// TIA Portal project "zadanie_2_Kral_dzvonar" (V15.1)

(* hardware
DEVICE "S7-1200 station_1"  S7-1200 Station
   slot 0: "Rack_0"  S7-1200 Rack  Rack  V1.0
   slot 1: "PLC_1"  CPU 1215C DC/DC/DC  6ES7 215-1AG40-0XB0  V4.3
*)

// ===== PLC "PLC_1"  CPU 1215C DC/DC/DC =====

VAR_GLOBAL   // PLC tag table "Default tag table"
   "OS1" AT %I0.4 : Bool;
   "OS2" AT %I0.5 : Bool;
   "OS3" AT %I0.7 : Bool;
   "OS4" AT %I1.0 : Bool;
   "KS5" AT %I0.6 : Bool;
   "KS2" AT %I0.1 : Bool;
   "KS1" AT %I0.0 : Bool;
   "KS4" AT %I0.2 : Bool;
   "KS3" AT %I0.3 : Bool;
   "P1_vzad" AT %Q0.0 : Bool;
   "P1_vpred" AT %Q0.1 : Bool;
   "P2_vpred" AT %Q0.2 : Bool;
   "P2_vzad" AT %Q0.3 : Bool;
   "S1" AT %Q0.6 : Bool;
   "S2" AT %Q1.0 : Bool;
   "D1" AT %Q0.4 : Bool;
   "D2" AT %Q0.5 : Bool;
   "D3" AT %Q0.7 : Bool;
   "D4" AT %Q1.1 : Bool;
   "pom" AT %M5.0 : Bool;
   "start" AT %M5.1 : Bool;
   "pom2" AT %M5.2 : Bool;
   "casOneskorenia" AT %MD6 : Time;
END_VAR

DATA_BLOCK "Dopravnik1"   // DB1
{ S7_Optimized_Access := 'TRUE' }
VERSION : 0.1
// stored: InstanceOfName Dopravnik
"Dopravnik"
BEGIN
END_DATA_BLOCK

DATA_BLOCK "ID"   // DB2
{ S7_Optimized_Access := 'TRUE' }
VERSION : 0.1
   VAR RETAIN
      id : Int := 3;
   END_VAR
BEGIN
END_DATA_BLOCK

DATA_BLOCK "Posuvac1"   // DB3
{ S7_Optimized_Access := 'TRUE' }
VERSION : 0.1
// stored: InstanceOfName Posuvac
"Posuvac"
BEGIN
END_DATA_BLOCK

DATA_BLOCK "Dopravnik2"   // DB4
{ S7_Optimized_Access := 'TRUE' }
VERSION : 0.1
// stored: InstanceOfName Dopravnik
"Dopravnik"
BEGIN
END_DATA_BLOCK

DATA_BLOCK "Stroj1"   // DB5
{ S7_Optimized_Access := 'TRUE' }
VERSION : 0.1
// stored: InstanceOfName stroj
"stroj"
BEGIN
END_DATA_BLOCK

DATA_BLOCK "Dopravnik3"   // DB6
{ S7_Optimized_Access := 'TRUE' }
VERSION : 0.1
// stored: InstanceOfName Dopravnik
"Dopravnik"
BEGIN
END_DATA_BLOCK

DATA_BLOCK "Stroj2"   // DB7
{ S7_Optimized_Access := 'TRUE' }
VERSION : 0.1
// stored: InstanceOfName stroj
"stroj"
BEGIN
END_DATA_BLOCK

DATA_BLOCK "Dopravnik4"   // DB8
{ S7_Optimized_Access := 'TRUE' }
VERSION : 0.1
// stored: InstanceOfName Dopravnik
"Dopravnik"
BEGIN
END_DATA_BLOCK

DATA_BLOCK "Posuvac2"   // DB10
{ S7_Optimized_Access := 'TRUE' }
VERSION : 0.1
// stored: InstanceOfName Posuvac
"Posuvac"
BEGIN
END_DATA_BLOCK

FUNCTION_BLOCK "Dopravnik"   // FB1, LAD
{ S7_Optimized_Access := 'TRUE' }
VERSION : 0.1
   VAR_INPUT
      predchadzajuci : Bool;
      aktualny : Bool;
      nasledujuci : Bool;
      input_id : Int;
      blok : Bool;
      resetFull : Bool;
      Cas : Time := T#500ms;
      oneskorenie : Bool;
   END_VAR
   VAR_OUTPUT
      chod : Bool;
   END_VAR
   VAR
      pom1 : Bool;
      pom2 : Bool;
      pom5 : Bool;
      pom3 : Bool;
      id : Int;
      full : Bool;
      oneskorenyBeh : Bool;
      IEC_Timer_0_Instance : TON_TIME;
      oneskorenyReset : Bool;
      IEC_Timer_0_Instance_1 : TON_TIME;
   END_VAR
   VAR_TEMP   // added for the SCL form of the ladder/FBD networks
      _w1 : Bool;
      _w2 : Bool;
   END_VAR
BEGIN

REGION Network 1
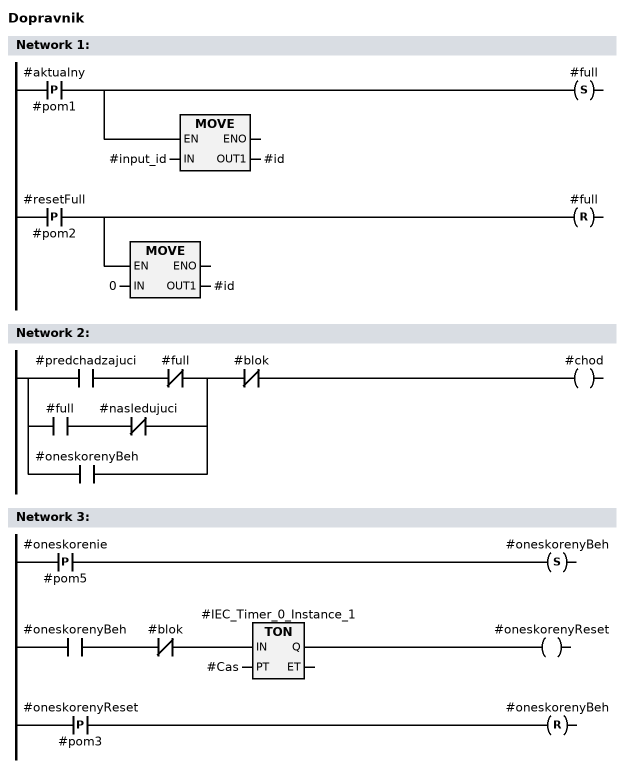
   RUNG wire#powerrail
      P_Contact(operand := #aktualny, bit := #pom1)
      wire#w1
      S_Coil( #full )
   END_RUNG
   RUNG wire#w1
      Move(in := #input_id, out1 => #id)
   END_RUNG
   RUNG wire#powerrail
      P_Contact(operand := #resetFull, bit := #pom2)
      wire#w2
      R_Coil( #full )
   END_RUNG
   RUNG wire#w2
      Move(in := 0, out1 => #id)
   END_RUNG
   // the same network as SCL:
   #_w1 := #aktualny AND NOT #pom1;   // rising edge of #aktualny
   #pom1 := #aktualny;
   IF #_w1 THEN
       #full := TRUE;
       #id := #input_id;
   END_IF;
   #_w2 := #resetFull AND NOT #pom2;   // rising edge of #resetFull
   #pom2 := #resetFull;
   IF #_w2 THEN
       #full := FALSE;
       #id := 0;
   END_IF;
END_REGION

REGION Network 2
   RUNG wire#powerrail
      Contact( #predchadzajuci )
      I_Contact( #full )
      wire#w1
      I_Contact( #blok )
      Coil( #chod )
   END_RUNG
   RUNG wire#powerrail
      Contact( #full )
      I_Contact( #nasledujuci )
   END_RUNG wire#w1
   RUNG wire#powerrail
      Contact( #oneskorenyBeh )
   END_RUNG wire#w1
   // the same network as SCL:
   #chod := ((#predchadzajuci AND NOT #full) OR (#full AND NOT #nasledujuci) OR #oneskorenyBeh) AND NOT #blok;
END_REGION

REGION Network 3
   #_w1 := #oneskorenie AND NOT #pom5;   // rising edge of #oneskorenie
   #pom5 := #oneskorenie;
   IF #_w1 THEN #oneskorenyBeh := TRUE; END_IF;
   #IEC_Timer_0_Instance_1(IN := #oneskorenyBeh AND NOT #blok, PT := #Cas);   // TON
   #oneskorenyReset := #IEC_Timer_0_Instance_1.Q;
   #_w2 := #oneskorenyReset AND NOT #pom3;   // rising edge of #oneskorenyReset
   #pom3 := #oneskorenyReset;
   IF #_w2 THEN #oneskorenyBeh := FALSE; END_IF;
END_REGION
END_FUNCTION_BLOCK

FUNCTION_BLOCK "stroj"   // FB2, LAD
{ S7_Optimized_Access := 'TRUE' }
VERSION : 0.1
   VAR_INPUT
      enable : Bool;
      N : Int;
      resetDopracoval : Bool;
   END_VAR
   VAR_OUTPUT
      pracuj : Bool;
   END_VAR
   VAR
      cas_prace : Time := T#2s;
      cas_prestoja : Time := T#1s;
      pracuje : Bool;
      Stroj_timer1 : TON_TIME;
      Stroj_timer2 : TON_TIME;
   END_VAR
   VAR RETAIN
      counter1 : CTU_INT;
      pom : Bool;
   END_VAR
   VAR
      dopracoval : Bool;
      pom2 : Bool;
   END_VAR
   VAR_TEMP   // added for the SCL form of the ladder/FBD networks
      _w1 : Bool;
      _w2 : Bool;
   END_VAR
BEGIN

REGION Network 1
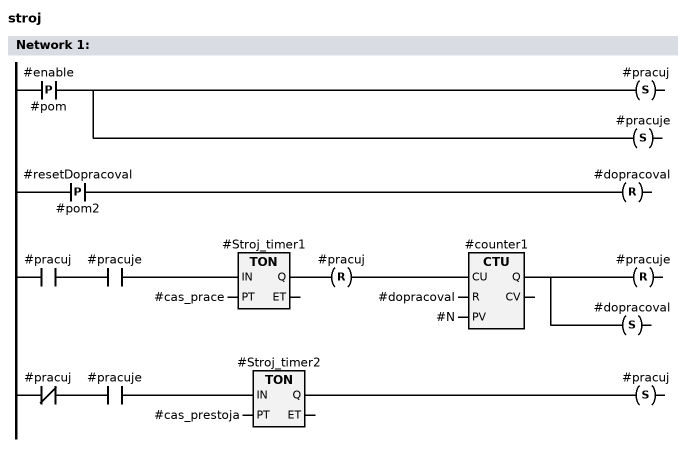
   #_w1 := #enable AND NOT #pom;   // rising edge of #enable
   #pom := #enable;
   IF #_w1 THEN
       #pracuj := TRUE;
       #pracuje := TRUE;
   END_IF;
   #_w2 := #resetDopracoval AND NOT #pom2;   // rising edge of #resetDopracoval
   #pom2 := #resetDopracoval;
   IF #_w2 THEN #dopracoval := FALSE; END_IF;
   #Stroj_timer1(IN := #pracuj AND #pracuje, PT := #cas_prace);   // TON
   IF #Stroj_timer1.Q THEN #pracuj := FALSE; END_IF;
   #counter1(CU := #Stroj_timer1.Q, R := #dopracoval, PV := #N);   // CTU
   IF #counter1.Q THEN
       #pracuje := FALSE;
       #dopracoval := TRUE;
   END_IF;
   #Stroj_timer2(IN := NOT #pracuj AND #pracuje, PT := #cas_prestoja);   // TON
   IF #Stroj_timer2.Q THEN #pracuj := TRUE; END_IF;
END_REGION
END_FUNCTION_BLOCK

FUNCTION_BLOCK "Posuvac"   // FB3, LAD
{ S7_Optimized_Access := 'TRUE' }
VERSION : 0.1
   VAR_INPUT
      stavVpredu : Bool;
      stavVzadu : Bool;
      enable : Bool;
      loading_time : Time;
      input_id : Int;
      posuvacVzad : Bool;
      posuvacVpred : Bool;
      resetFull : Bool;
   END_VAR
   VAR_OUTPUT
      vpred : Bool;
      vzad : Bool;
   END_VAR
   VAR
      pom1 : Bool;
      pom5 : Bool;
      loading : Bool;
      id : Int;
      IEC_Timer_0_Instance : TON_TIME;
      full : Bool;
      done : Bool;
   END_VAR
   VAR_TEMP   // added for the SCL form of the ladder/FBD networks
      _w1 : Bool;
   END_VAR
BEGIN

REGION Network 1
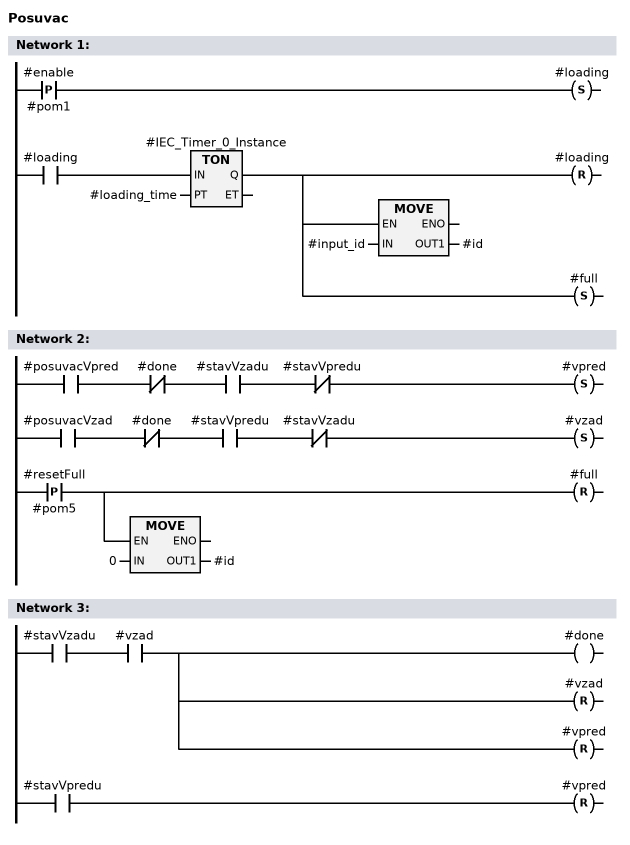
   #_w1 := #enable AND NOT #pom1;   // rising edge of #enable
   #pom1 := #enable;
   IF #_w1 THEN #loading := TRUE; END_IF;
   #IEC_Timer_0_Instance(IN := #loading, PT := #loading_time);   // TON
   IF #IEC_Timer_0_Instance.Q THEN
       #loading := FALSE;
       #id := #input_id;
       #full := TRUE;
   END_IF;
END_REGION

REGION Network 2
   RUNG wire#powerrail
      Contact( #posuvacVpred )
      I_Contact( #done )
      Contact( #stavVzadu )
      I_Contact( #stavVpredu )
      S_Coil( #vpred )
   END_RUNG
   RUNG wire#powerrail
      Contact( #posuvacVzad )
      I_Contact( #done )
      Contact( #stavVpredu )
      I_Contact( #stavVzadu )
      S_Coil( #vzad )
   END_RUNG
   RUNG wire#powerrail
      P_Contact(operand := #resetFull, bit := #pom5)
      wire#w1
      R_Coil( #full )
   END_RUNG
   RUNG wire#w1
      Move(in := 0, out1 => #id)
   END_RUNG
   // the same network as SCL:
   IF #posuvacVpred AND NOT #done AND #stavVzadu AND NOT #stavVpredu THEN #vpred := TRUE; END_IF;
   IF #posuvacVzad AND NOT #done AND #stavVpredu AND NOT #stavVzadu THEN #vzad := TRUE; END_IF;
   #_w1 := #resetFull AND NOT #pom5;   // rising edge of #resetFull
   #pom5 := #resetFull;
   IF #_w1 THEN
       #full := FALSE;
       #id := 0;
   END_IF;
END_REGION

REGION Network 3
   RUNG wire#powerrail
      Contact( #stavVzadu )
      Contact( #vzad )
      wire#w1
      Coil( #done )
   END_RUNG
   RUNG wire#w1
      R_Coil( #vzad )
   END_RUNG
   RUNG wire#w1
      R_Coil( #vpred )
   END_RUNG
   RUNG wire#powerrail
      Contact( #stavVpredu )
      R_Coil( #vpred )
   END_RUNG
   // the same network as SCL:
   #done := #stavVzadu AND #vzad;
   IF #done THEN
       #vzad := FALSE;
       #vpred := FALSE;
   END_IF;
   IF #stavVpredu THEN #vpred := FALSE; END_IF;
END_REGION
END_FUNCTION_BLOCK

ORGANIZATION_BLOCK "Main"   // OB1, LAD, ProgramCycle
TITLE = "Main Program Sweep (Cycle)"
{ S7_Optimized_Access := 'TRUE' }
VERSION : 0.1
   VAR_INPUT
      Initial_Call : Bool;   // Initial call of this OB
      Remanence : Bool;   // =True, if remanent data are available
   END_VAR
   VAR_TEMP   // added for the SCL form of the ladder/FBD networks
      _w1 : Bool;
      _w2 : Bool;
   END_VAR
BEGIN

REGION Network 1
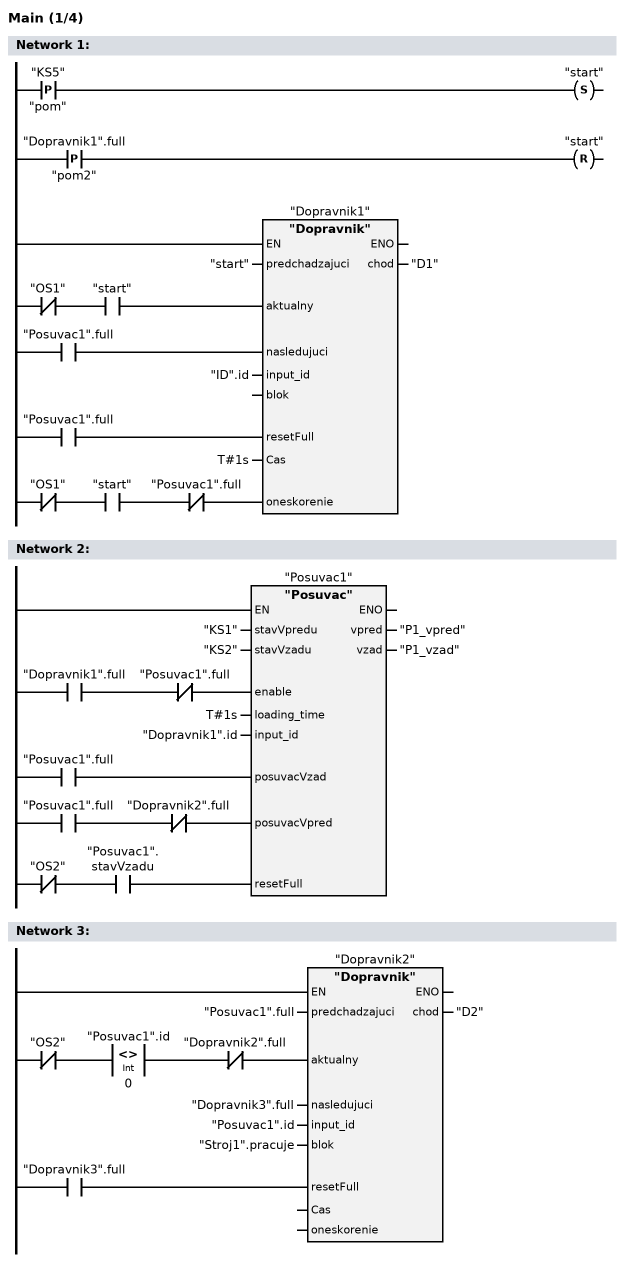
   RUNG wire#powerrail
      P_Contact(operand := "KS5", bit := "pom")
      S_Coil( "start" )
   END_RUNG
   RUNG wire#powerrail
      P_Contact(operand := "Dopravnik1".full, bit := "pom2")
      R_Coil( "start" )
   END_RUNG
   RUNG wire#powerrail
      "Dopravnik1"(aktualny := wire#w1, nasledujuci := wire#w2, resetFull := wire#w3, oneskorenie := wire#w4, predchadzajuci := "start", input_id := "ID".id, blok :=, Cas := T#1s, chod => "D1")
   END_RUNG
   RUNG wire#powerrail
      I_Contact( "OS1" )
      Contact( "start" )
   END_RUNG wire#w1
   RUNG wire#powerrail
      Contact( "Posuvac1".full )
   END_RUNG wire#w2
   RUNG wire#powerrail
      Contact( "Posuvac1".full )
   END_RUNG wire#w3
   RUNG wire#powerrail
      I_Contact( "OS1" )
      Contact( "start" )
      I_Contact( "Posuvac1".full )
   END_RUNG wire#w4
   // the same network as SCL:
   #_w1 := "KS5" AND NOT "pom";   // rising edge of "KS5"
   "pom" := "KS5";
   IF #_w1 THEN "start" := TRUE; END_IF;
   #_w2 := "Dopravnik1".full AND NOT "pom2";   // rising edge of "Dopravnik1".full
   "pom2" := "Dopravnik1".full;
   IF #_w2 THEN "start" := FALSE; END_IF;
   "Dopravnik1"(predchadzajuci := "start",   // "Dopravnik"
                aktualny := NOT "OS1" AND "start",
                nasledujuci := "Posuvac1".full,
                input_id := "ID".id,
                resetFull := "Posuvac1".full,
                Cas := T#1s,
                oneskorenie := NOT "OS1" AND "start" AND NOT "Posuvac1".full,
                chod => "D1");
END_REGION

REGION Network 2
   RUNG wire#powerrail
      "Posuvac1"(enable := wire#w1, posuvacVzad := wire#w2, posuvacVpred := wire#w3, resetFull := wire#w4, stavVpredu := "KS1", stavVzadu := "KS2", loading_time := T#1s, input_id := "Dopravnik1".id, vpred => "P1_vpred", vzad => "P1_vzad")
   END_RUNG
   RUNG wire#powerrail
      Contact( "Dopravnik1".full )
      I_Contact( "Posuvac1".full )
   END_RUNG wire#w1
   RUNG wire#powerrail
      Contact( "Posuvac1".full )
   END_RUNG wire#w2
   RUNG wire#powerrail
      Contact( "Posuvac1".full )
      I_Contact( "Dopravnik2".full )
   END_RUNG wire#w3
   RUNG wire#powerrail
      I_Contact( "OS2" )
      Contact( "Posuvac1".stavVzadu )
   END_RUNG wire#w4
   // the same network as SCL:
   "Posuvac1"(stavVpredu := "KS1",   // "Posuvac"
              stavVzadu := "KS2",
              enable := "Dopravnik1".full AND NOT "Posuvac1".full,
              loading_time := T#1s,
              input_id := "Dopravnik1".id,
              posuvacVzad := "Posuvac1".full,
              posuvacVpred := "Posuvac1".full AND NOT "Dopravnik2".full,
              resetFull := NOT "OS2" AND "Posuvac1".stavVzadu,
              vpred => "P1_vpred",
              vzad => "P1_vzad");
END_REGION

REGION Network 3
   RUNG wire#powerrail
      "Dopravnik2"(aktualny := wire#w1, resetFull := wire#w2, predchadzajuci := "Posuvac1".full, nasledujuci := "Dopravnik3".full, input_id := "Posuvac1".id, blok := "Stroj1".pracuje, Cas :=, oneskorenie :=, chod => "D2")
   END_RUNG
   RUNG wire#powerrail
      I_Contact( "OS2" )
      { S7_Templates := "SrcType := Int" } NE_Contact(in1 := "Posuvac1".id, in2 := 0)
      I_Contact( "Dopravnik2".full )
   END_RUNG wire#w1
   RUNG wire#powerrail
      Contact( "Dopravnik3".full )
   END_RUNG wire#w2
   // the same network as SCL:
   "Dopravnik2"(predchadzajuci := "Posuvac1".full,   // "Dopravnik"
                aktualny := NOT "OS2" AND ("Posuvac1".id <> 0) AND NOT "Dopravnik2".full,
                nasledujuci := "Dopravnik3".full,
                input_id := "Posuvac1".id,
                blok := "Stroj1".pracuje,
                resetFull := "Dopravnik3".full,
                chod => "D2");
END_REGION

REGION Network 4
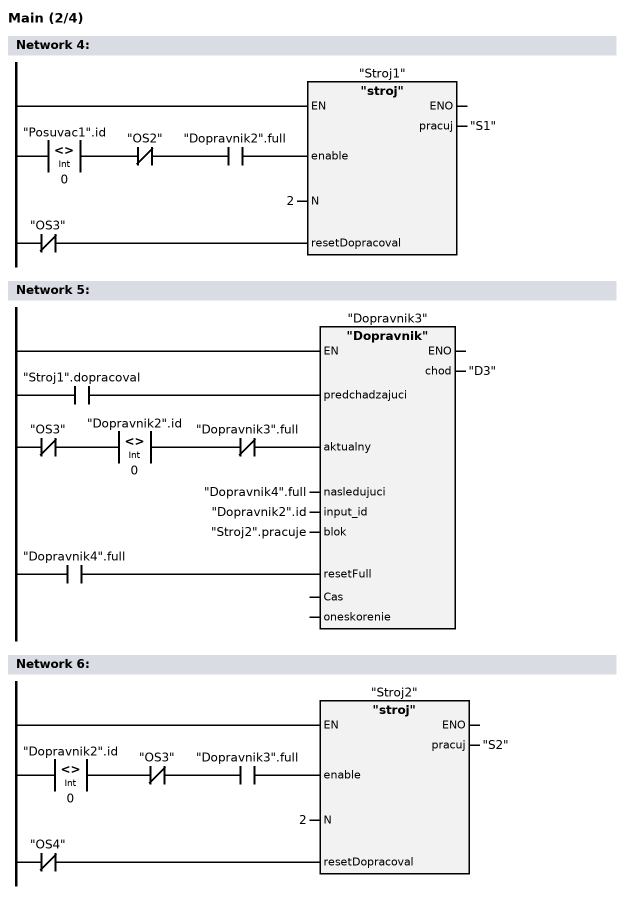
   RUNG wire#powerrail
      "Stroj1"(enable := wire#w1, resetDopracoval := wire#w2, N := 2, pracuj => "S1")
   END_RUNG
   RUNG wire#powerrail
      { S7_Templates := "SrcType := Int" } NE_Contact(in1 := "Posuvac1".id, in2 := 0)
      I_Contact( "OS2" )
      Contact( "Dopravnik2".full )
   END_RUNG wire#w1
   RUNG wire#powerrail
      I_Contact( "OS3" )
   END_RUNG wire#w2
   // the same network as SCL:
   "Stroj1"(enable := ("Posuvac1".id <> 0) AND NOT "OS2" AND "Dopravnik2".full,   // "stroj"
            N := 2,
            resetDopracoval := NOT "OS3",
            pracuj => "S1");
END_REGION

REGION Network 5
   RUNG wire#powerrail
      "Dopravnik3"(predchadzajuci := wire#w1, aktualny := wire#w2, resetFull := wire#w3, nasledujuci := "Dopravnik4".full, input_id := "Dopravnik2".id, blok := "Stroj2".pracuje, Cas :=, oneskorenie :=, chod => "D3")
   END_RUNG
   RUNG wire#powerrail
      Contact( "Stroj1".dopracoval )
   END_RUNG wire#w1
   RUNG wire#powerrail
      I_Contact( "OS3" )
      { S7_Templates := "SrcType := Int" } NE_Contact(in1 := "Dopravnik2".id, in2 := 0)
      I_Contact( "Dopravnik3".full )
   END_RUNG wire#w2
   RUNG wire#powerrail
      Contact( "Dopravnik4".full )
   END_RUNG wire#w3
   // the same network as SCL:
   "Dopravnik3"(predchadzajuci := "Stroj1".dopracoval,   // "Dopravnik"
                aktualny := NOT "OS3" AND ("Dopravnik2".id <> 0) AND NOT "Dopravnik3".full,
                nasledujuci := "Dopravnik4".full,
                input_id := "Dopravnik2".id,
                blok := "Stroj2".pracuje,
                resetFull := "Dopravnik4".full,
                chod => "D3");
END_REGION

REGION Network 6
   RUNG wire#powerrail
      "Stroj2"(enable := wire#w1, resetDopracoval := wire#w2, N := 2, pracuj => "S2")
   END_RUNG
   RUNG wire#powerrail
      { S7_Templates := "SrcType := Int" } NE_Contact(in1 := "Dopravnik2".id, in2 := 0)
      I_Contact( "OS3" )
      Contact( "Dopravnik3".full )
   END_RUNG wire#w1
   RUNG wire#powerrail
      I_Contact( "OS4" )
   END_RUNG wire#w2
   // the same network as SCL:
   "Stroj2"(enable := ("Dopravnik2".id <> 0) AND NOT "OS3" AND "Dopravnik3".full,   // "stroj"
            N := 2,
            resetDopracoval := NOT "OS4",
            pracuj => "S2");
END_REGION

REGION Network 7
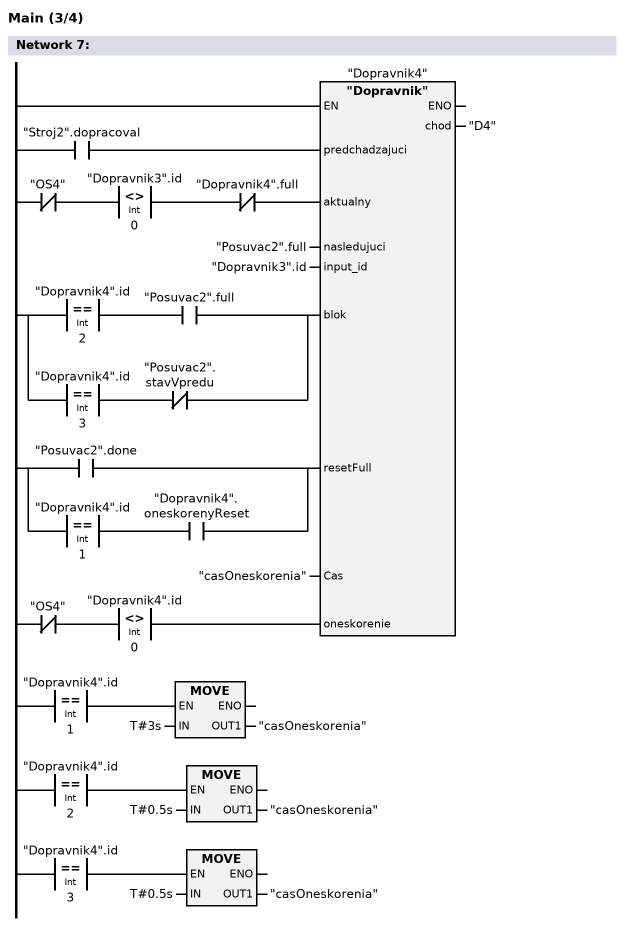
   RUNG wire#powerrail
      "Dopravnik4"(predchadzajuci := wire#w1, aktualny := wire#w2, blok := wire#w3, resetFull := wire#w4, oneskorenie := wire#w5, nasledujuci := "Posuvac2".full, input_id := "Dopravnik3".id, Cas := "casOneskorenia", chod => "D4")
   END_RUNG
   RUNG wire#powerrail
      Contact( "Stroj2".dopracoval )
   END_RUNG wire#w1
   RUNG wire#powerrail
      I_Contact( "OS4" )
      { S7_Templates := "SrcType := Int" } NE_Contact(in1 := "Dopravnik3".id, in2 := 0)
      I_Contact( "Dopravnik4".full )
   END_RUNG wire#w2
   RUNG wire#powerrail
      { S7_Templates := "SrcType := Int" } EQ_Contact(in1 := "Dopravnik4".id, in2 := 2)
      Contact( "Posuvac2".full )
   END_RUNG wire#w3
   RUNG wire#powerrail
      { S7_Templates := "SrcType := Int" } EQ_Contact(in1 := "Dopravnik4".id, in2 := 3)
      I_Contact( "Posuvac2".stavVpredu )
   END_RUNG wire#w3
   RUNG wire#powerrail
      Contact( "Posuvac2".done )
   END_RUNG wire#w4
   RUNG wire#powerrail
      { S7_Templates := "SrcType := Int" } EQ_Contact(in1 := "Dopravnik4".id, in2 := 1)
      Contact( "Dopravnik4".oneskorenyReset )
   END_RUNG wire#w4
   RUNG wire#powerrail
      I_Contact( "OS4" )
      { S7_Templates := "SrcType := Int" } NE_Contact(in1 := "Dopravnik4".id, in2 := 0)
   END_RUNG wire#w5
   RUNG wire#powerrail
      { S7_Templates := "SrcType := Int" } EQ_Contact(in1 := "Dopravnik4".id, in2 := 1)
      Move(in := T#3s, out1 => "casOneskorenia")
   END_RUNG
   RUNG wire#powerrail
      { S7_Templates := "SrcType := Int" } EQ_Contact(in1 := "Dopravnik4".id, in2 := 2)
      Move(in := T#0.5s, out1 => "casOneskorenia")
   END_RUNG
   RUNG wire#powerrail
      { S7_Templates := "SrcType := Int" } EQ_Contact(in1 := "Dopravnik4".id, in2 := 3)
      Move(in := T#0.5s, out1 => "casOneskorenia")
   END_RUNG
   // the same network as SCL:
   "Dopravnik4"(predchadzajuci := "Stroj2".dopracoval,   // "Dopravnik"
                aktualny := NOT "OS4" AND ("Dopravnik3".id <> 0) AND NOT "Dopravnik4".full,
                nasledujuci := "Posuvac2".full,
                input_id := "Dopravnik3".id,
                blok := (("Dopravnik4".id = 2) AND "Posuvac2".full) OR (("Dopravnik4".id = 3) AND NOT "Posuvac2".stavVpredu),
                resetFull := "Posuvac2".done OR (("Dopravnik4".id = 1) AND "Dopravnik4".oneskorenyReset),
                Cas := "casOneskorenia",
                oneskorenie := NOT "OS4" AND ("Dopravnik4".id <> 0),
                chod => "D4");
   IF "Dopravnik4".id = 1 THEN "casOneskorenia" := T#3s; END_IF;
   IF "Dopravnik4".id = 2 THEN "casOneskorenia" := T#0.5s; END_IF;
   IF "Dopravnik4".id = 3 THEN "casOneskorenia" := T#0.5s; END_IF;
END_REGION

REGION Network 8
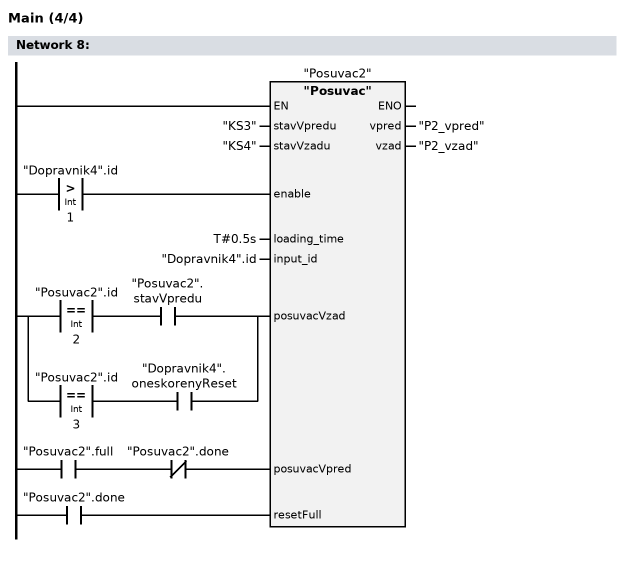
   RUNG wire#powerrail
      "Posuvac2"(enable := wire#w1, posuvacVzad := wire#w2, posuvacVpred := wire#w3, resetFull := wire#w4, stavVpredu := "KS3", stavVzadu := "KS4", loading_time := T#0.5s, input_id := "Dopravnik4".id, vpred => "P2_vpred", vzad => "P2_vzad")
   END_RUNG
   RUNG wire#powerrail
      { S7_Templates := "SrcType := Int" } GT_Contact(in1 := "Dopravnik4".id, in2 := 1)
   END_RUNG wire#w1
   RUNG wire#powerrail
      { S7_Templates := "SrcType := Int" } EQ_Contact(in1 := "Posuvac2".id, in2 := 2)
      Contact( "Posuvac2".stavVpredu )
   END_RUNG wire#w2
   RUNG wire#powerrail
      { S7_Templates := "SrcType := Int" } EQ_Contact(in1 := "Posuvac2".id, in2 := 3)
      Contact( "Dopravnik4".oneskorenyReset )
   END_RUNG wire#w2
   RUNG wire#powerrail
      Contact( "Posuvac2".full )
      I_Contact( "Posuvac2".done )
   END_RUNG wire#w3
   RUNG wire#powerrail
      Contact( "Posuvac2".done )
   END_RUNG wire#w4
   // the same network as SCL:
   "Posuvac2"(stavVpredu := "KS3",   // "Posuvac"
              stavVzadu := "KS4",
              enable := "Dopravnik4".id > 1,
              loading_time := T#0.5s,
              input_id := "Dopravnik4".id,
              posuvacVzad := (("Posuvac2".id = 2) AND "Posuvac2".stavVpredu) OR (("Posuvac2".id = 3) AND "Dopravnik4".oneskorenyReset),
              posuvacVpred := "Posuvac2".full AND NOT "Posuvac2".done,
              resetFull := "Posuvac2".done,
              vpred => "P2_vpred",
              vzad => "P2_vzad");
END_REGION
END_ORGANIZATION_BLOCK